// TwinCAT 3 PLC project PLCproject
// ProgramVersion: 3.1.4024.0
// libraries:
//   Tc2_MC2, * (Beckhoff Automation GmbH)
//   Tc2_Standard, * (Beckhoff Automation GmbH)
//   Tc2_System, * (Beckhoff Automation GmbH)
//   Tc3_Module, * (Beckhoff Automation GmbH)
// project tree:
//   / PlcTask.TcTTO
//   POUs/ MAIN.TcPOU
// real-time tasks:
//   TASK PlcTask: cycle T#10ms, priority 20, ADS port 350
// motion (NC):
//   TASK NC-Task 1 SAF: cycle T#2ms, priority 4, ADS port 501
//   TASK NC-Task 1 SVB: cycle T#10ms, priority 8, ADS port 511
//   AXIS Axis 1 (id 1)
//     OtherSettings: AllowMotionCmdToSlave=true
//     encoder EncType=4
//       EncPara: MaxCount=#x0000ffff
//         Inc: RefSoftSyncMask=#x0000ffff
//     drive DrvType=24
//       Analog: TorqueSetpointScale=10, ScaleFactorActTorque=0.1
//       TimeComp: TaskDelayCycles=1
//     controller CtrType=1
//       CtrPara: PriorControlFactor=1
//         Observer: BandWidth=20
//   AXIS Axis 2 (id 2)
//     OtherSettings: AllowMotionCmdToSlave=true
//     encoder EncType=19
//       EncPara: MaxCount=#xffffffff
//     drive DrvType=16
//       DrvPara: MaxCount=#xffffffff, DriveControlDWord=#x00020000
//         Analog: TorqueSetpointScale=10, ScaleFactorActTorque=0.1
//         TimeComp: TaskDelayCycles=1
//     controller CtrType=1
//       CtrPara: PriorControlFactor=1
//         Observer: BandWidth=20
//   AXIS Axis 3 (id 3)
//     OtherSettings: AllowMotionCmdToSlave=true
//     encoder EncType=8
//       EncPara: MaxCount=#xffffffff
//     drive DrvType=9
//       DrvPara: MaxCount=#xffffffff, DriveControlDWord=#x00030100
//         Analog: VeloScale=1.02400649589962, TorqueSetpointScale=10, ScaleFactorActTorque=0.1
//         TimeComp: TaskDelayCycles=1
//     controller CtrType=1
//       CtrPara: PriorControlFactor=1
//         Observer: BandWidth=20
//   AXIS Axis 4 (id 4)
//     OtherSettings: AllowMotionCmdToSlave=true
//     encoder EncType=8
//       EncPara: MaxCount=#xffffffff
//     drive DrvType=9
//       DrvPara: MaxCount=#xffffffff, DriveControlDWord=#x00030100
//         Analog: VeloScale=1.02400649589962, TorqueSetpointScale=10, ScaleFactorActTorque=0.1
//         TimeComp: TaskDelayCycles=1
//     controller CtrType=1
//       CtrPara: PriorControlFactor=1
//         Observer: BandWidth=20
// I/O:
//   DEVICE Device 1 (EtherCAT), AmsNetId 169.254.190.45.2.1
//     Term 1 (EK1200) [EK1200-5000 EtherCAT Power supply (2A E-Bus)]
//       Term 2 (EL1008) [EL1008 8Ch. Dig. Input 24V, 3ms]
//       Term 3 (EL2008) [EL2008 8Ch. Dig. Output 24V, 0.5A]
//       Term 4 (EL5151) [EL5151 1Ch. Inc. Encoder]
//       Term 5 (EL9110) [EL9110 Power Supplier with LED (24V, Diagnostics)]
//       Term 6 (EL9576) [EL9576 Brake chopper terminal]
//       Term 7 (EL7037) [EL7037 1Ch. Stepper motor output stage (24V, 1.5A)]
//       Term 8 (EL9512) [EL9512 Power supply terminal 12V]
//       Term 9 (EL3162) [EL3162 2Ch. Ana. Input 0-10V]
//       Term 10 (EL4102) [EL4102 2Ch. Ana. Output  0-10V, 16bit]
//       Term 11 (EL6910) [EL6910, TwinSAFE PLC]
//       Term 12 (EK1122) [EK1122 2 port EtherCAT junction]
//         Term 13 (EK1100) [EK1100 EtherCAT Coupler (2A E-Bus)]
//           Term 14 (EL1859) [EL1859 8Ch. Dig. Input 24V, 3ms, 8Ch. Dig. Output 24V, 0.5A]
//           Term 15 (EL1904) [EL1904, 4 Ch. Safety Input 24V, TwinSAFE]
//             modules: Module 1 (FSOES)
//           Term 16 (EL2904) [EL2904, 4 Ch. Safety Output 24V, 0.5A, TwinSAFE]
//             modules: Module 1 (FSOES), Module 2 (DO)
//           Term 17 (EL9110) [EL9110 Power Supplier with LED (24V, Diagnostics)]
//           Term 18 (EL2004) [EL2004 4Ch. Dig. Output 24V, 0.5A]
//           Term 19 (EL9410) [EL9410 E-Bus Power Supplier  (Diagnostics)]
//           Term 20 (EL7201-9014) [EL7201-9014 1Ch. MDP742 Servo motor output stage with OCT (50V, 2.8A RMS) and STO input]
//           Term 29 (EL9011) [EL9011 End Terminal]
//         Term 21 (EK1101) [EK1101 EtherCAT Coupler (2A E-Bus, ID switch)]
//           Term 22 (EL1904) [EL1904, 4 Ch. Safety Input 24V, TwinSAFE]
//             modules: Module 1 (FSOES)
//           Term 23 (EL1252) [EL1252 2Ch. Fast Dig. Input 24V, 1µs, DC Latch]
//           Term 24 (EL1262) [EL1262 2Ch. Dig. Input 24V, 1µs, DC Oversample]
//           Term 25 (EL2252) [EL2252 2Ch. Dig. Output 24V, 0.5A, DC Time Stamp]
//           Term 26 (EL3702) [EL3702 2Ch. Ana. Input +/-10V, DIFF, Oversample]
//           Term 27 (EL4732) [EL4732 2Ch. Ana. Output +/-10V, Oversample]
//           Term 30 (EL9011) [EL9011 End Terminal]
//         Drive 28 (AX5203-0000-0210) [AX5203-0000-0210 EtherCAT Drive (SoE, 2 Ch.)]
// variable links:
//   NC-Task 1 SAF/Axes/Axis 1 <-> Device 1 (EtherCAT)/Term 1 (EK1200)/Term 7 (EL7037)
//     Drive/Inputs/In/nState1 @bit 3 <-> STM Status/Status/Error
//     Drive/Inputs/In/nState1 @bit 7 <-> STM Status/Status/Motor stall
//     Drive/Inputs/In/nState1 @bit 5 <-> STM Status/Status/Moving negative
//     Drive/Inputs/In/nState1 @bit 4 <-> STM Status/Status/Moving positive
//     Drive/Inputs/In/nState1 @bit 1 <-> STM Status/Status/Ready
//     Drive/Inputs/In/nState1 <-> STM Status/Status/Ready to enable
//     Drive/Inputs/In/nState1 @bit 6 <-> STM Status/Status/Torque reduced
//     Drive/Inputs/In/nState1 @bit 2 <-> STM Status/Status/Warning
//     Drive/Inputs/In/nState2 @bit 3 <-> STM Status/Status/Digital input 1
//     Drive/Inputs/In/nState2 @bit 4 <-> STM Status/Status/Digital input 2
//     Drive/Inputs/In/nState2 @bit 5 <-> STM Status/Status/Sync error
//     Drive/Inputs/In/nState2 @bit 7 <-> STM Status/Status/TxPDO Toggle
//     Drive/Inputs/In/nState4 @bit 1 <-> WcState/InputToggle
//     Drive/Inputs/In/nState4 <-> WcState/WcState
//     Drive/Outputs/Out/nCtrl1 <-> STM Control/Control/Enable
//     Drive/Outputs/Out/nCtrl1 @bit 2 <-> STM Control/Control/Reduce torque
//     Drive/Outputs/Out/nCtrl1 @bit 1 <-> STM Control/Control/Reset
//     Drive/Outputs/Out/nCtrl2 @bit 3 <-> STM Control/Control/Digital output 1
//     Drive/Outputs/Out/nDataOut2[0] <-> STM Velocity/Velocity
//     Enc/Inputs/In/nDataIn1[0] <-> ENC Status compact/Counter value
//     Enc/Inputs/In/nDataIn2[0] <-> ENC Status compact/Latch value
//     Enc/Inputs/In/nState1 @bit 4 <-> ENC Status compact/Status/Counter overflow
//     Enc/Inputs/In/nState1 @bit 3 <-> ENC Status compact/Status/Counter underflow
//     Enc/Inputs/In/nState1 @bit 7 <-> ENC Status compact/Status/Extrapolation stall
//     Enc/Inputs/In/nState1 <-> ENC Status compact/Status/Latch C valid
//     Enc/Inputs/In/nState1 @bit 1 <-> ENC Status compact/Status/Latch extern valid
//     Enc/Inputs/In/nState1 @bit 2 <-> ENC Status compact/Status/Set counter done
//     Enc/Inputs/In/nState2 @bit 4 <-> ENC Status compact/Status/Status of extern latch
//     Enc/Inputs/In/nState2 <-> ENC Status compact/Status/Status of input A
//     Enc/Inputs/In/nState2 @bit 1 <-> ENC Status compact/Status/Status of input B
//     Enc/Inputs/In/nState2 @bit 2 <-> ENC Status compact/Status/Status of input C
//     Enc/Inputs/In/nState2 @bit 5 <-> ENC Status compact/Status/Sync error
//     Enc/Inputs/In/nState2 @bit 7 <-> ENC Status compact/Status/TxPDO Toggle
//     Enc/Inputs/In/nState4 @bit 1 <-> WcState/InputToggle
//     Enc/Inputs/In/nState4 <-> WcState/WcState
//     Enc/Outputs/Out/nCtrl1 <-> ENC Control compact/Control/Enable latch C
//     Enc/Outputs/Out/nCtrl1 @bit 3 <-> ENC Control compact/Control/Enable latch extern on negative edge
//     Enc/Outputs/Out/nCtrl1 @bit 1 <-> ENC Control compact/Control/Enable latch extern on positive edge
//     Enc/Outputs/Out/nCtrl1 @bit 2 <-> ENC Control compact/Control/Set counter
//     Enc/Outputs/Out/nDataOut1[0] <-> ENC Control compact/Set counter value
//   NC-Task 1 SAF/Axes/Axis 2 <-> Device 1 (EtherCAT)/Term 1 (EK1200)/Term 12 (EK1122)/Term 13 (EK1100)/Term 20 (EL7201-9014)
//     Drive/Inputs/In/nDcOutputTime <-> InfoData/DcOutputShift
//     Drive/Inputs/In/nState1 <-> DRV Statusword/Statusword
//     Drive/Inputs/In/nState2 <-> DRV Statusword/Statusword @bit 8
//     Drive/Inputs/In/nState4 @bit 1 <-> WcState/InputToggle
//     Drive/Inputs/In/nState4 <-> WcState/WcState
//     Drive/Outputs/Out/nCtrl1 <-> DRV Controlword/Controlword
//     Drive/Outputs/Out/nCtrl2 <-> DRV Controlword/Controlword @bit 8
//     Drive/Outputs/Out/nDataOut2 <-> DRV Target velocity/Target velocity
//     Enc/Inputs/In/nDataIn1 <-> FB Position/Position
//     Enc/Inputs/In/nDcInputTime <-> InfoData/DcInputShift
//     Enc/Inputs/In/nState4 @bit 1 <-> WcState/InputToggle
//     Enc/Inputs/In/nState4 <-> WcState/WcState
//   NC-Task 1 SAF/Axes/Axis 3 <-> Device 1 (EtherCAT)/Term 1 (EK1200)/Term 12 (EK1122)/Drive 28 (AX5203-0000-0210)
//     Drive/Inputs/In/nDataIn1 <-> AT 1/Following distance
//     Drive/Inputs/In/nDcOutputTime <-> InfoData/DcOutputShift
//     Drive/Inputs/In/nState1 <-> AT 1/Drive status word @bit 8
//     Drive/Inputs/In/nState2 <-> AT 1/Drive status word
//     Drive/Inputs/In/nState4 @bit 1 <-> WcState/InputToggle
//     Drive/Inputs/In/nState4 <-> WcState/WcState
//     Drive/Outputs/Out/nCtrl1 <-> MDT 1/Master control word @bit 8
//     Drive/Outputs/Out/nDataOut1 <-> MDT 1/Position command value
//     Enc/Inputs/In/nDataIn1 <-> AT 1/Position feedback 1 value
//     Enc/Inputs/In/nDcInputTime <-> InfoData/DcInputShift
//     Enc/Inputs/In/nState4 @bit 1 <-> WcState/InputToggle
//     Enc/Inputs/In/nState4 <-> WcState/WcState
//   NC-Task 1 SAF/Axes/Axis 4 <-> Device 1 (EtherCAT)/Term 1 (EK1200)/Term 12 (EK1122)/Drive 28 (AX5203-0000-0210)
//     Drive/Inputs/In/nDataIn1 <-> AT 2/Following distance
//     Drive/Inputs/In/nDcOutputTime <-> InfoData/DcOutputShift
//     Drive/Inputs/In/nState1 <-> AT 2/Drive status word @bit 8
//     Drive/Inputs/In/nState2 <-> AT 2/Drive status word
//     Drive/Inputs/In/nState4 @bit 1 <-> WcState/InputToggle
//     Drive/Inputs/In/nState4 <-> WcState/WcState
//     Drive/Outputs/Out/nCtrl1 <-> MDT 2/Master control word @bit 8
//     Drive/Outputs/Out/nDataOut1 <-> MDT 2/Position command value
//     Enc/Inputs/In/nDataIn1 <-> AT 2/Position feedback 1 value
//     Enc/Inputs/In/nDcInputTime <-> InfoData/DcInputShift
//     Enc/Inputs/In/nState4 @bit 1 <-> WcState/InputToggle
//     Enc/Inputs/In/nState4 <-> WcState/WcState
//   PLCproject/PLCproject Instance <-> Device 1 (EtherCAT)/Term 1 (EK1200)/Term 2 (EL1008)
//     PlcTask Inputs/MAIN.bHalt <-> Channel 4/Input
//     PlcTask Inputs/MAIN.bMotorEnable <-> Channel 1/Input
//     PlcTask Inputs/MAIN.bVelocity1 <-> Channel 2/Input
//     PlcTask Inputs/MAIN.bVelocity2 <-> Channel 3/Input
//   PLCproject/PLCproject Instance <-> Device 1 (EtherCAT)/Term 1 (EK1200)/Term 3 (EL2008)
//     PlcTask Outputs/MAIN.bLED{1..4} <-> Channel {1..4}/Output  (4 links)
//   PLCproject/PLCproject Instance <-> NC-Task 1 SAF/Axes/Axis 4
//     PlcTask Inputs/MAIN.BottomRightMotor.NcToPlc <-> Outputs/ToPlc
//     PlcTask Outputs/MAIN.BottomRightMotor.PlcToNc <-> Inputs/FromPlc

CONFIGURATION PLCproject
    RESOURCE PLC ON TwinCAT3
        TASK PlcTask(INTERVAL := T#10ms, PRIORITY := 20);
        PROGRAM MAIN WITH PlcTask : MAIN;
    END_RESOURCE
END_CONFIGURATION

// ---- POUs/MAIN.TcPOU
PROGRAM MAIN
VAR
	bMotorEnable, bVelocity1, bVelocity2, bHalt	AT %I* 	: BOOL;
	bLED1, bLED2, bLED3, bLED4					AT %Q*	: BOOL;
	xEnable												: BOOL;
	
	BottomRightMotor			: AXIS_REF;
	fbMC_Power 					: MC_Power;
	fbMC_Velocity				: MC_MoveVelocity;
	fbMC_Halt					: MC_Halt;
END_VAR

IF bMotorEnable THEN
	xEnable := TRUE;
	bLED1	:= TRUE; //turns on LED above switch
ELSE
	xEnable := FALSE;
	bLED1	:= FALSE;//turns on LED above switch
END_IF

fbMC_Power(
	Axis:=BottomRightMotor,
	Enable:=xEnable,
	Enable_Positive:=xEnable,
	Enable_Negative:=xEnable,
	Override:=100.0);
	
fbMC_Velocity(
	Axis:=BottomRightMotor,
	Execute:=bVelocity1,
	Velocity:= 100.0);	
	
fbMC_Velocity(
	Axis:=BottomRightMotor,
	Execute:=bVelocity2,
	Velocity:= 400.0);	
	
fbMC_Halt(
	Axis:=BottomRightMotor,
	Execute:= bHalt);
	
	
//--------------------
//  LEDs
IF bVelocity1 THEN
	bLED2	:= TRUE; //turns on LED above switch
ELSE
	bLED2	:= FALSE;//turns on LED above switch
END_IF

IF bVelocity2 THEN
	bLED3	:= TRUE; //turns on LED above switch
ELSE
	bLED3	:= FALSE;//turns on LED above switch
END_IF

IF bHalt THEN
	bLED4	:= TRUE; //turns on LED above switch
ELSE
	bLED4	:= FALSE;//turns on LED above switch
END_IF

END_PROGRAM
